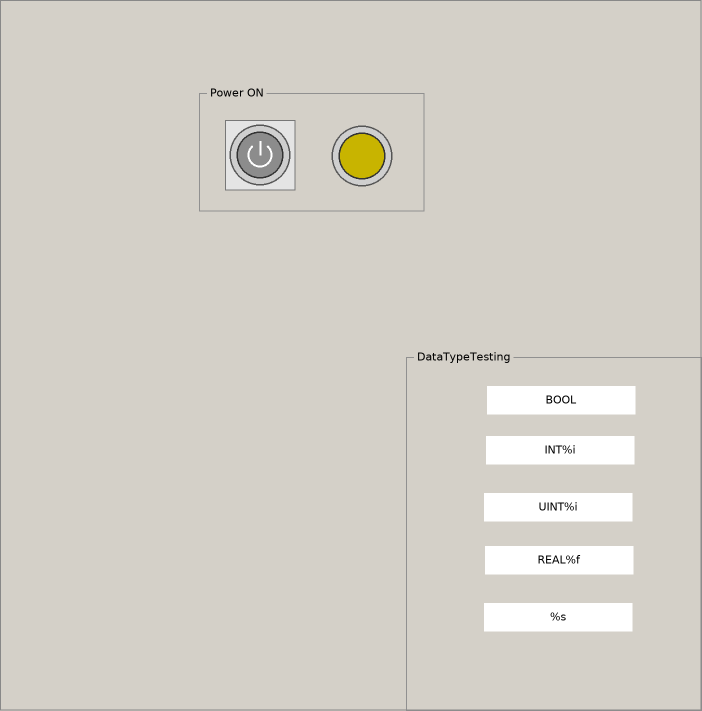
VISUALIZATION Visualization  // 702x711
    GroupBox (199,85 225x126), "Power ON"
        Lamp1 (128,36 70x70), variable: MAIN.bEnable, style: Lamp-Lamp1-Yellow
        PowerSwitch (26,35 70x70), variable: MAIN.bStart, behaviour: TOGGLE, style: Switch-PowerSwitch-Gray
    GroupBox (406,349 296x362), "DataTypeTesting"
        Textfield (80,36 150x30), "BOOL"
        Textfield (79,86 150x30), "INT%i", text variable: MAIN.nINT
        Textfield (77,143 150x30), "UINT%i", text variable: MAIN.nUINT
        Textfield (78,196 150x30), "REAL%f", text variable: MAIN.fREAL
            OnMouseDown: write the text variable via Default
        Textfield (77,253 150x30), "%s", text variable: MAIN.sPowerStatus
            OnMouseDown: write the text variable via Default
END_VISUALIZATION

(* stored: Version 1.1.0.1, ProductVersion 3.1.4024.12
   Visu Visualization: Id {cc1c38df-e33c-4951-bdb8-9c3bd4f4d4d6} *)
